PROGRAM MAIN
VAR
	fbTimeObj: FB_TIME;
	fbTimerObj: FB_TIMER;
	
	
END_VAR

fbTimeObj();

fbTimerObj(fbTimerRef := fbTimeObj);

END_PROGRAM

(* stored: Version 1.1.0.1, ProductVersion 3.1.4024.11
   POU MAIN: Id {0da3a7ac-0d35-4c21-8d5f-ea439bb447f7}, SpecialFunc None *)
